(* CoDeSys 2.3 export: export.EXP *)

(* Global variable list: UserGlobals/Globals *)
VAR_GLOBAL
    G_SafeInvertTest : INT := 0;
END_VAR

(* Data type in UserTypes *)
TYPE
    TestStruct : STRUCT
        Value   : INT := 0;
        IsValid : BOOL := FALSE;
        Name    : STRING := '';
    END_STRUCT;

    TestEnum : (
        stIdle   := 0,
        stactive := 1,
        stError  := 2
    );
END_TYPE

(* POU SafeInvert, ST *)
FUNCTION SafeInvert : INT
VAR_INPUT
    value : INT;
END_VAR
IF value = -32768 THEN
    SafeInvert := 32767;
ELSE
    SafeInvert := 0 - value;
END_IF;
END_FUNCTION
